// TIA Portal V20 export
// export: Created 2025-12-01T14:56:17.7542577Z, ExportSetting None, DisplayName Totally Integrated Automation Portal, DisplayVersion V20 Update 3, DisplayName TIA Portal Openness, DisplayVersion V20 Update 3, DisplayName TIA Portal Version Control Interface, DisplayVersion V20 Update 3, DisplayName STEP 7 Professional, DisplayVersion V20 Update 3, DisplayName STEP 7 Safety, DisplayVersion V20 Update 2, DisplayName WinCC Basic/Comfort/Advanced, DisplayVersion V20 Update 3, DisplayName WinCC Professional, DisplayVersion V20 Update 3, DisplayName WinCC Unified, DisplayVersion V20 Update 3
TYPE "TipoMesaPantalla"
   STRUCT
      Tipo_Mesa : USInt := 50;   // Define el numero de la pantalla a lanzar cuando pulsemos sobre el boton de la mesa
      Tipo_interlock : USInt := 0;   // Define el numero de interlock a mostrar. si es 0 no hay interlock
      Phs_1 : Bool;   // Define si hay que mostrar la fotocelula 1
      Phs_2 : Bool;   // Define si hay que mostrar la fotocelula 2
      Phs_3 : Bool;   // Define si hay que mostrar la fotocelula 3
      Phs_4 : Bool;   // Define si hay que mostrar la fotocelula 4
      Phs_5 : Bool;   // Define si hay que mostrar la fotocelula 5
      Byte2_bit5 : Bool;   // --libre--
      Byte2_bit6 : Bool;   // --libre--
      Byte2_bit7 : Bool := 0;   // --libre--
      Protusion_1 : Bool;   // Define si hay que mostrar la protusion 1
      Protusion_2 : Bool;   // Define si hay que mostrar la protusion 2
      Protusion_3 : Bool;   // Define si hay que mostrar la protusion 3
      Protusion_4 : Bool;   // Define si hay que mostrar la protusion 4
      Byte3_bit4 : Bool;   // --libre--
      Detector_carretilla : Bool;   // Define si hay que mostrar el detector de carretilla
      Byte3_bit6 : Bool;   // --libre--
      Byte3_bit7 : Bool := 0;   // --libre--
      Rodillos : Bool;   // Define si el transportador tiene rodillos
      Cadenas : Bool;   // Define si el transportador tiene cadenas
      Transfer : Bool;   // Define si el transportador tiene transfer
      Tope_1 : Bool;   // Define si el transportador tiene tope 1
      Tope_2 : Bool;   // Define si el transportador tiene tope 2
      Giro : Bool;   // Define si el transportador tiene mesa de giro
      Bidireccional_rodillos : Bool;   // Define si el transportador es bidireccional en rodillos
      Bidireccional_cadenas : Bool;   // Define si el transportador es bidireccional en correas
      Byte5_bit0 : Bool;   // --libre--
      Byte5_bit1 : Bool;   // --libre--
      Byte5_bit2 : Bool;   // --libre--
      Byte5_bit3 : Bool;   // --libre--
      Byte5_bit4 : Bool;   // --libre--
      Byte5_bit5 : Bool;   // --libre--
      PermisoDeModificar : Bool;   // Define si el transportador tiene que pedir permiso para modificar los datos de las UTs
      Byte5_bit7 : Bool;   // --libre--
      Tipo_maquina : UInt;   // Define el numero de pantalla a lanzar cuando tenemos maquina. a cero no muestra ninguna
   END_STRUCT;
END_TYPE
